Universal Robots PolyScope program: rtde_control_loop.urp

Program rtde_control_loop (installation=default directory=/ursim/programs createdIn=3.2.19275 lastSavedIn=5.19.0 robotSerialNumber=20195599999)
Calibrated DH parameters: a=[0, -0.425, -0.3922, 0, 0, 0]; d=[0.1625, 0, 0, 0.1333, 0.0997, 0.0996]; alpha=[1.570796, 0, 0, 1.570796, -1.570796, 0]; deltaTheta=[0, 0, 0, 0, 0, 0]
InitVariablesNode
BeforeStart
  setp := p[0,0,0,0,0,0]
  SuppressedNode
    Script: rtde_set_watchdog("input_int_register_0", 1, "PAUSE")
  Script: write_output_integer_register(0, 1)
Robot Program (runOnlyOnce=false)
  If read_input_integer_register(0)≟1 and setp≠p[0, 0, 0, 0, 0, 0]
    'Valid pose received from client'
    MoveL speed 80 mm/s, acceleration 400 mm/s^2 (useActiveTCP=true) feature=Base
      Waypoint Variable (Variable): variable=setp
    'Confirm that move was executed'
    Script: write_output_integer_register(0, 0)
    'Wait until script acknowledges confirmation'
    Loop While (checkContinuously=false) expression=read_input_integer_register(0)≟1
      Script: sync()
    'Request next pose'
    Script: write_output_integer_register(0, 1)
  Script: sync()
Thread Thread_1 (runOnlyOnce=false)
  Loop Forever
    tmp := p[0,0,0,0,0,0]
    Script: tmp[0] = read_input_float_register(0)
    Script: tmp[1] = read_input_float_register(1)
    Script: tmp[2] = read_input_float_register(2)
    Script: tmp[3] = read_input_float_register(3)
    Script: tmp[4] = read_input_float_register(4)
    Script: tmp[5] = read_input_float_register(5)
    setp := tmp
    Script: sync()
